
// ===== library types =====

// folder: LIOLink

TYPE "LIOLink_typeDiagnostics"
   STRUCT
      status : Word;   // Status of the Block or error identification when error occurred
      subfunctionStatus : DWord;   // Status or return value of called FB's, FCs and system blocks
      stateNumber : DInt;   // State in the state machine of the block where the error occurred
   END_STRUCT;
END_TYPE

// folder: iJaw

TYPE "UDT_iJawDataRcv"
   STRUCT
      Gauge1 : Word;   // ADC Eingang der Sensorrohdaten (min.: 0 max.: 4096)
      Gauge2 : Word;   // ADC Eingang der Sensorrohdaten (min.: 0 max.: 4096)
      Battery : Byte;   // Rohsignal aktuelle Batteriespannung (min.: 0 .. max.: 157) [V]
      Temperature : Byte;   // Rohsignal Temperatursensor (min.: -40 .. max.: 125) [°C]
      GyroXaxis : Byte;   // Rohsignal Beschleunigungssensor X (min.: -128 .. max.: 127) [g]
      GyroYaxis : Byte;   // Rohsignal Beschleunigungssensor Y (min.: -128 .. max.: 127) [g]
      GyroZaxis : Byte;   // Rohsignal Beschleunigungssensor Z (min.: -128 .. max.: 127) [g]
      Warning : Byte;   // Warnungs-/Fehlercode (Bit0:= Klemmkraft überschritten; Bit1:= Klemmkraft unters
      Force1 : Word;   // Spannkraft Kanal 1 (min.: 0 .. max.: 65,535) [N]
      Force2 : Word;   // Spannkraft Kanal 2 (min.: 0 .. max.: 65,535) [N]
      Reserve1431 : Array[14..31] of Byte;   // Reserve
   END_STRUCT;
END_TYPE

TYPE "UDT_iJawDataSend"
   STRUCT
      nRotSpeedSpindleAct : Int;   // actual rotational speed of the spindle
      pHydCylChamber1Act : Byte;   // actual hydraulic pressure in actuating cylinder chamber for outer clamping
      pHydCylChamber2Act : Byte;   // actual hydraulic pressure in actuating cylinder chamber for outer clamping
      AHydCylChamber1Act : Byte;   // hydraulic area of cylinder chamber for outer clamping
      AHydCylChamber2Act : Byte;   // hydraulic area of cylinder chamber for outer clamping
      Reserve0631 : Array[6..31] of Byte;   // Reserve
   END_STRUCT;
END_TYPE

TYPE "UDT_iJawDataSendUser"
VERSION : 0.1
   STRUCT
      RelCmdSysMode : Bool;   // Trigger sende Kommando change System Mode (see Mode)
      RelCmdTara : Bool;   // Trigger sende Kommando Tara
      RelReadType : Bool;   // Trigger sende Kommando lese iJaw Type
      RelIMA : Bool;   // Trigger sende Kommando IMA
      RelForceTreshold : Bool;   // Trigger sende Kommando Force Treshold
      RelNoiseLevel : Bool;   // Trigger sende Kommando Noise Level
      RelStoreToFlash : Bool;   // Trigger sende Kommando Store to Flash
      NoiseLevel : UInt;   // Höhe der Kraftänderung innerhalb der Samplerate 100Hz, die zur Bestimmung einer Messdatenübertragung neben dem Schwellwert herangezogen wird.
      ForceTreshold : UDInt;   // Schwellwert der Spannkraftsumme die anliegt, um im Mode 2 kontinuierlich Daten zu übertragen
      IMA : USInt;   // Zeitintervall in s, innerhalb der die iJaw spätestens einen neuen Messwert an den Empfänger überträgt
      Mode : Byte;   // Select Mode (0x1 = continuous mode; 0x2 = state dependent mode
      nRotSpeedSpindleAct : Int;   // actual rotational speed of the spindle
      pHydCylChamber1Act : Byte;   // actual hydraulic pressure in actuating cylinder chamber for outer clamping
      pHydCylChamber2Act : Byte;   // actual hydraulic pressure in actuating cylinder chamber for outer clamping
      AHydCylChamber1Act : Byte;   // hydraulic area of cylinder chamber for outer clamping
      AHydCylChamber2Act : Byte;   // hydraulic area of cylinder chamber for outer clamping
   END_STRUCT;
END_TYPE

TYPE "UDT_iJawDataRcvUser"
VERSION : 0.1
   STRUCT
      Gauge1 : UInt;   // ADC Eingang der Sensorrohdaten (min.: 0 max.: 4096)
      Gauge2 : UInt;   // ADC Eingang der Sensorrohdaten (min.: 0 max.: 4096)
      Battery : USInt;   // Rohsignal aktuelle Batteriespannung (min.: 0 .. max.: 157) [V]
      Temperature : SInt;   // Rohsignal Temperatursensor (min.: -40 .. max.: 125) [°C]
      GyroXaxis : SInt;   // Rohsignal Beschleunigungssensor X (min.: -128 .. max.: 127) [g]
      GyroYaxis : SInt;   // Rohsignal Beschleunigungssensor Y (min.: -128 .. max.: 127) [g]
      GyroZaxis : SInt;   // Rohsignal Beschleunigungssensor Z (min.: -128 .. max.: 127) [g]
      Warning : Byte;   // Warnungs-/Fehlercode (Bit0:= Klemmkraft überschritten; Bit1:= Klemmkraft unters
      Force1 : UInt;   // Spannkraft Kanal 1 (min.: 0 .. max.: 65,535) [N]
      Force2 : UInt;   // Spannkraft Kanal 2 (min.: 0 .. max.: 65,535) [N]
      iJawType : String;   // Ausgelesen Typ des iJaws
   END_STRUCT;
END_TYPE

TYPE "UDT_iJawIOFifo"
   STRUCT
      cmd : USInt;   // kommando
      isuCmdData : "UDT_iJawISDUCmdData";
   END_STRUCT;
END_TYPE

TYPE "UDT_iJawISDUCmdData"
TITLE = UDT_iJawISDUCmdData
// Command daten für die isdu / io-link kommunikation
   STRUCT
      execute : Bool;   // Anforderung zum Ausführen der Funktion
      readWrite : Bool;   // FALSE: lesen, TRUE: schreiben
      port : Int;   // Port am IO-Link-Master-Modul
      index : Int;   // Adressparameterindex (IO-Link Device); 0..32767: IOL-D; 65535: Portfunktionen
      subindex : Int;   // Adressparameter Subindex (IO-Link Device); 0: vollständige Aufzeichnung; 1-255: Einzelparameter
      writeLen : Int;   // Länge der Schreibdaten (Nettodaten); 1..232
   END_STRUCT;
END_TYPE

// folder: (top level)

FUNCTION "GetHwDevice" : Int   // FC1, SCL
TITLE = GetHwDevice
{ S7_Optimized_Access := 'TRUE' }
AUTHOR : HeitecAg
VERSION : 0.1
// Ermitteln einer Hardware-Kennung eines DP-Slaves/PROFINET IO-Devices anhand einer E/A-Adresse
   VAR_INPUT
      varEaAdresse : Variant;   // EA-Adresse (E, A, PE, PA) innerhalb eines Moduls.
   END_VAR
   VAR_OUTPUT
      hwDevice : HW_DEVICE;   // Ermittelte Hardware-Kennung eines DP-Slaves/PROFINET IO-Devices
   END_VAR
   VAR_TEMP
      thwAny : HW_ANY;   // Ermittelte Hardware-Kennung (logische Adresse) des EA-Moduls.
      tgeoAdr : GEOADDR;   // Geografische Adresse
   END_VAR
   // Ret_Val : Fehlercode der Anweisungen.
   VAR CONSTANT
      DEF_HE_DEVICE : HW_DEVICE := 0;   // Initalwert für output hw_device
      HWTYPE : UInt := 2;   // Hardwaretyp: 2: IO-Device / DP-Slave
      SLOT : UInt := 0;   // Steckplatz-Nummer
      SUB_SLOT : UInt := 0;   // Nummer des Submoduls. Falls kein Submodul vorhanden ist oder gesteckt werden kann, hat dieser Parameter den Wert "0".
   END_VAR
BEGIN
   REGION BLOCK INFO HEADER
     //==========================================================================================================
     //Title:        GetHwDevice
     //Function:     Ermitteln einer Hardware-Kennung eines DP-Slaves/PROFINET IO-Devices anhand einer E/A-Adresse
     //----------------------------------------------------------------------------------------------------------
     //Change log table:
     //Version       | Date          | Expert in charge      | Changes applied
     //----------------------------------------------------------------------------------------------------------
     //1.0.0         | 26.06.23      | HeitecAg                | First released Version
     //==========================================================================================================
   END_REGION BLOCK INFO HEADER

   #hwDevice := #DEF_HE_DEVICE;

   #GetHwDevice := IO2MOD(ADDR := #varEaAdresse, LADDR => #thwAny);

   IF (#GetHwDevice = 0)THEN
     #GetHwDevice := LOG2GEO(LADDR := #thwAny, GEOADDR := #tgeoAdr);
   END_IF;

   IF (#GetHwDevice = 0) THEN
     #tgeoAdr.HWTYPE := #HWTYPE;
     #tgeoAdr.SLOT := 0;
     #tgeoAdr.SUBSLOT := 0;

     #GetHwDevice := GEO2LOG(GEOADDR := #tgeoAdr, LADDR => #hwDevice);
   END_IF;

   ENO := (#GetHwDevice = 0);
   RETURN;
END_FUNCTION

// folder: LIOLink/S7-1200/1500/Base blocks

FUNCTION_BLOCK "LIOLink_Device"   // FB50004, SCL
TITLE = LIOLink_Device / LIOLINK_DEVICE
{ S7_Optimized_Access := 'TRUE' }
AUTHOR : SIOS
FAMILY : LIOLink
VERSION : 4.0
// Acyclically reads or writes data records from and to IO-Link devices / Funktionsbaustein zum Lesen und Schreiben von azyklischen Daten auf Geräten mit IO-Link, die auf SIMATIC S7-Steuerungen verwendet werden. (früher IO_LINK_CALL)
   VAR_INPUT
      execute : Bool;   // Request to execute function / Anforderung zum Ausführen der Funktion
      hwID : HW_IO;   // Hardware identifier of IO-Link master module or first sub module / Hardware-Kennung des IO-Link-Mastermoduls (Submodul für ET 200eco PN)
      cap : Int;   // Client Access Point (CAP) 0xB400 or 0x00E3 (227) / Client Access Point (CAP); 0xB400 für ET 200eco PN, CM 8x IO-Link, sonst 0xE003 (227)
      readWrite : Bool;   // FALSE: read-mode, TRUE: write-mode / FALSE: lesen, TRUE: schreiben
      port : Int;   // Port on IO-Link master module / Port am IO-Link-Master-Modul
      index : Int;   // Address parameter index (IO-Link device); 0..32767: IOL-D; 65535: port functions / Adressparameterindex (IO-Link Device); 0..32767: IOL-D; 65535: Portfunktionen
      subindex : Int;   // Address parameter subindex (IO-Link device); 0: full record; 1-255: single parameter / Adressparameter Subindex (IO-Link Device); 0: vollständige Aufzeichnung; 1-255: Einzelparameter
      writeLen : Int;   // Length of writing data (net data); 1..232 / Länge der Schreibdaten (Nettodaten); 1..232
      timeout : Time := T#20S;   // Time after which the request is aborted / Zeit, nach der die Anfrage abgebrochen wird
      pollingPeriod : Time := T#100MS;   // Time period of polling
   END_VAR
   VAR_OUTPUT
      done : Bool;   // TRUE: FB processing successfully completed / TRUE: FB-Bearbeitung erfolgreich abgeschlossen
      busy : Bool;   // TRUE: FB is active and new output values can be expected. / TRUE: FB ist aktiv und neue Ausgangswerte sind zu erwarten.
      error : Bool;   // FALSE: No error / TRUE: An error occurred during the execution of the FB. / FALSE: Kein Fehler / TRUE: Bei der Ausführung des FB ist ein Fehler aufgetreten.
      status : Word := 16#7000;   // 16#0000-16#7FFF: Status of the FB / 16#8000-16#FFFF: Error identification (see following table) / 16#0000-16#7FFF: Status des FB / 16#8000-16#FFFF: Fehleridentifikation (siehe folgende Tabelle)
      diagnostics : "LIOLink_typeDiagnostics";   // Diagnostics information of FB / Diagnoseinformationen der FB
      readLen : Int;   // Length of read data record (number of bytes) / Länge des gelesenen Datensatzes (Anzahl Bytes)
   END_VAR
   VAR_IN_OUT
      record : Array[*] of Byte;   // Data area for reading/writing data (max. 232 byte) / Datenbereich zum Lesen/Schreiben von Daten (max. 232 Byte)
   END_VAR
   VAR
      statExecuteOld : Bool;   // Old value of 'execute' input for edge detection / Alter Wert des 'Execute'-Eingangs für Flankenerkennung
      statDone : Bool;   // Static value for output 'done' / Statischer Wert für Ausgang 'done'
      statBusy : Bool;   // Static value for output 'busy' / Statischer Wert für Ausgang 'besetzt'
      statError : Bool;   // Static value for output 'error' / Statischer Wert für Ausgang 'error'
      statStatus : Word := 16#7000;   // Static value for output 'status' / Statischer Wert für Ausgang 'Status'
      statPollingPeriod : Time := T#100MS;   // Static value for input 'pollingPeriod'
      statHwID : HW_IO;   // Static value for input 'hwID' / Statischer Wert für Eingang 'hwID'
      statHwIDprevious : HW_IO;   // Static value for input 'hwID' from the previous execute / Statischer Wert für Eingang 'hwID'
      statReadWrite : Bool;   // Static value for input 'readWrite' / Stativwert für Eingabe 'readWrite'
      statCap : UInt;   // Static value for input 'cap' / Statischer Wert für Eingabe 'cap'
      statTimeout : Time;   // Static value for input 'timeout' / Statischer Wert für Eingang 'timeout'
      statLen : UInt;   // Length of data to be written to device / Länge der Daten, die auf das Gerät geschrieben werden sollen
      statSubfunctionStatus : DWord;   // Status of WRREC/RDREC or error code from IO-Link Master (%W1: IO-Link Master error, %W0: ISDU error) / Status von WRREC/RDREC oder Fehlercode vom IO-Link-Master (%W1: IO-Link-Master-Fehler, %W0: ISDU-Fehler)
      statFBErrorState : DInt;   // State in the state machine of the block where the error occurred / Zustand in der Zustandsmaschine des Blocks, in dem der Fehler aufgetreten ist
      statFBState : DInt := 0;   // State in the state machine of the FB / Zustand in der Zustandsmaschine der FB
      statEmptyDiagnostics : "LIOLink_typeDiagnostics";   // Empty diagnostics information (for initialization purposes only) / Leere Diagnoseinformationen (nur für Initialisierungszwecke)
      instRdRec : RDREC;   // System function "read data record" / Systemfunktion "Datensatz lesen"
      instWrRec : WRREC;   // System function "write data record" / Systemfunktion "Datensatz schreiben"
      instPoll : TP_TIME;   // poll rate read data record / Abfragerate Datensatz lesen
      instMonitor : TON_TIME;   // request monitoring time / Überwachungszeit anfordern
      statRead : Struct   // data area for reading data / Datenbereich zum Lesen von Daten
         header : Struct   // Header
            call : Struct   // header for read/write data record / Header für Datensatz lesen/schreiben
               extFunctionNum : Byte := 16#08;   // extended function number (fix coded 08h) / erweiterte Funktionsnummer (fix codiert 08h)
               port : Byte;   // variable port (user interface) 0...255 / variabler Port (Benutzeroberfläche) 0...255
               fiIndex : Word := 16#FE4A;   // FI index (fix coded 65098) / FI-Index (fix codiert 65098)
            END_STRUCT;
            iolHeader : Struct   // header for IO-Link / Header für IO-Link
               control : Byte;   // RD_WR = 0 = read = Control:=0x03 / / RD_WR = 1 = write = Control:=0x02 / RD_WR = 0 = lesen = Steuerung:=0x03 / / RD_WR = 1 = schreiben = Steuerung:=0x02
               indexHighByte : Byte;   // index of data record 0…32767 (high byte) / Index des Datensatzes 0…32767 (High Byte)
               indexLowByte : Byte;   // index of data record 0…32767 (low byte) / Index des Datensatzes 0…32767 (Low Byte)
               subindex : Byte;   // subindex for data record 0...255 / Subindex für Datensatz 0...255
            END_STRUCT;
         END_STRUCT;
         data : Array[0..231] of Byte;   // Data
      END_STRUCT;
      statWrite : Struct   // data area for writing data / Datenbereich zum Schreiben von Daten
         header : Struct   // Header
            call : Struct   // header for read/write data record / Header für Datensatz lesen/schreiben
               extFunctionNum : Byte := 16#08;   // extended function number (fix coded 08h) / erweiterte Funktionsnummer (fix codiert 08h)
               port : Byte;   // variable port (user interface) 0...255 / variabler Port (Benutzeroberfläche) 0...255
               fiIndex : Word := 16#FE4A;   // FI index (fix coded 65098) / FI-Index (fix codiert 65098)
            END_STRUCT;
            iolHeader : Struct   // header für IO-Link / Header für IO-Link
               control : Byte;   // RD_WR = 0 = read = Control:=0x03 / / RD_WR = 1 = write = Control:=0x02 / RD_WR = 0 = lesen = Steuerung:=0x03 / / RD_WR = 1 = schreiben = Steuerung:=0x02
               indexHighByte : Byte;   // index of data record 0…32767 (high byte) / Index des Datensatzes 0…32767 (High Byte)
               indexLowByte : Byte;   // index of data record 0…32767 (low byte) / Index des Datensatzes 0…32767 (Low Byte)
               subindex : Byte;   // subindex for data record 0...255 / Subindex für Datensatz 0...255
            END_STRUCT;
         END_STRUCT;
         data : Array[0..231] of Byte;   // Data
      END_STRUCT;
   END_VAR
   VAR_TEMP
      tempExecute : Bool;   // Temporary value for input 'execute' / Temporärer Wert für Eingabe 'execute'
      tempHwID : HW_IO;   // Temporary value for input 'hwID'
      tempPort : Int;   // Temporary value for input 'port'
      tempIndex : Int;   // Temporary value for input 'index'
      tempSubindex : Int;   // Temporary value for input 'subindex'
      tempIndexCounter : DInt;   // run tag for counting loops / Run-Tag für Zählschleifen
   END_VAR
   VAR CONSTANT
      MODE_READ : Bool := FALSE;   // Mode to read data / Modus zum Lesen von Daten
      MODE_WRITE : Bool := TRUE;   // Mode to write data / Modus zum Schreiben von Daten
      MAX_PORT : USInt := 63;   // Max. possible port / max. möglichen Hafen
      MAX_INDEX : UInt := 32767;   // Max. possible index / max. möglicher Index
      INDEX_PORT_FUNC : UInt := 65535;   // Index to address port functions / Index zum Adressieren von Portfunktionen
      MAX_SUBINDEX : USInt := 255;   // Max. possible subindex / max. möglicher Subindex
      MAX_DATA : USInt := 232;   // Max. size of data to be transferred / max. Größe der zu übertragenden Daten
      UPPER_LIMIT : DInt := 231;   // Upper limit of data to be transferred / Obergrenze der zu übertragenden Daten
      FB_STATE_NO_PROCESSING : DInt := 0;   // FB state: No processing / FB-Zustand: Keine Verarbeitung
      FB_STATE_WRITE : DInt := 1;   // FB state: Write data record / Datensatz schreiben
      FB_STATE_POLL : DInt := 2;   // FB state: Wait and poll for response / warten und auf Antwort abfragen
      FB_STATE_READ_CAP : DInt := 3;   // FB state: Read cap / CAP lesen
      IOL_HEADER : UInt := 65098;   // Header IO-Link / Kopfzeile IO-Link
      LEN_HEADER : USInt := 8;   // Length of header / Länge des Headers
      CONTROL_WRITE : Byte := 16#02;   // Write data record / Datensatz schreiben
      CONTROL_READ : Byte := 16#03;   // Read data record / Datensatz lesen
      STATUS_EXECUTION_FINISHED : Word := 16#0000;   // Execution finished without errors / Ausführung ohne Fehler beendet
      STATUS_NO_CALL : Word := 16#7000;   // No job being currently processed / Derzeit wird kein Auftrag bearbeitet
      STATUS_FIRST_CALL : Word := 16#7001;   // First call after incoming new job (rising edge 'execute') / Erster Aufruf nach eingehendem neuen Auftrag (steigende Flanke 'execute')
      STATUS_SUBSEQUENT_CALL : Word := 16#7002;   // Subsequent call during active processing without further details / Nachfolgender Aufruf während aktiver Bearbeitung ohne weitere Angaben
      SUB_STATUS_NO_ERROR : Word := 16#0000;   // No error occured in subfunction call / Fehler: falscher Port
      ERR_WRONG_PORT : Word := 16#8201;   // Error: wrong port / Fehler: falscher Index
      ERR_WRONG_INDEX : Word := 16#8202;   // Error: wrong index / Fehler: falscher Subindex
      ERR_WRONG_SUBINDEX : Word := 16#8203;   // Error: wrong subindex / Fehler: falsche Länge für Datensatz schreiben
      ERR_WRONG_LENGTH : Word := 16#8205;   // Error: wrong length for write data record / Fehler: IO-Link-Master hat Fehlercode zurückgegeben, siehe "Diagnose"
      ERR_IO_LINK : Word := 16#8401;   // Error: IO-Link master returned error code, see "diagnostics" / Fehler: Gelesener Datensatz stimmt nicht mit Anfrage überein
      ERR_INCONSISTENT_DATA : Word := 16#8402;   // Error: Read data record doesn't match request / Fehler: Zeitüberschreitung bei Anforderung
      ERR_REQUEST_TIMEOUT : Word := 16#8403;   // Error: Request timed out / Fehler: Aufgrund eines undefinierten Zustands in der Zustandsmaschine
      ERR_UNDEFINED_STATE : Word := 16#8600;   // Error: due to an undefined state in state machine / Fehler: Aufgrund eines undefinierten Zustands in der Zustandsmaschine
      ERR_WRREC : Word := 16#8601;   // Error: WRREC encountered an error, see "diagnostics" / Fehler: WRREC hat einen Fehler festgestellt, siehe "Diagnose"
      ERR_RDREC : Word := 16#8602;   // Error: RDREC encountered an error, see "diagnostics" / Fehler: RDREC hat einen Fehler festgestellt, siehe "Diagnose"
      STATUS_MASK : DWord := 16#00FF_FF00;   // Mask to filter error codes / Maske zum Filtern von Fehlercodes
      STATUS_RESOURCE_BUSY : DWord := 16#0080_C200;   // Status from WRREC/RDREC: Resource is busy / Status von WRREC/RDREC: Ressource ist beschäftigt
      INDEX_CAP_IOLINK : Word := 16#B000;   // Index of the data record for IOLM_Info. Only IO-Link-Masters with CAP=16#B000 support this call. / Index des Datensatzes für IOLM_Info. Nur IO-Link-Master mit CAP=16#B000 unterstützen diesen Aufruf.
      CAP_LEGACY : Word := 16#00E3;   // Siemens (old) Standard CAP: 227 / Siemens (alt) Standard CAP: 227
      CAP_STANDARD : Word := 16#B400;   // IO-Link Standard CAP: 16#B400 / IO-Link-Standard-CAP: 16#B400
      STATUS_RDREC_VALID : Byte := 16#00;   // Status Code of RDREC in cased of no error occurs
      BITMASK_ERR_RDREC_B3 : Byte := 16#DE;   // Status Code of RDREC in case of an error when reading a data record
      BITMASK_ERR_RDREC_B2 : Byte := 16#80;   // Status Code of RDREC in case of an error when reading a data record - Error according to IEC 61158-6
      BITMASK_ERR_RDREC_B1 : Byte := 16#B0;   // Status Code of RDREC in case of an error when reading a data record - invalid index (cap)
   END_VAR
BEGIN
   REGION BLOCK INFO HEADER
       //===============================================================================
       // Siemens / (c)Copyright 2023
       //-------------------------------------------------------------------------------
       // Title:            LIOLink_Device
       // Function:         Acyclically reads or writes data records from and to IO-Link devices
       // Library:          LIOLink
       // Author:           Siemens Industry Online Support
       // Tested with:      CPU 1513-1 PN FW 2.8
       // Engineering:      TIA Portal V16
       // Restrictions:     S7-1200/1500
       // Requirements:     --
       //-------------------------------------------------------------------------------
       // Change log table:
       // Version  | Date       | Expert in charge       | Changes applied
       //----------|------------|------------------------|------------------------------
       // 02.00.00 | 30.09.2013 | Online Support         | First release for TIA Portal V12 SP1 as IO_LINK_CALL
       // 02.01.00 | 14.03.2014 | Online Support         | Upgrade to TIA Portal V13
       //                                                | Upgrade of system function 'WRREC' from V1.0 to V1.1
       // 03.00.00 | 28.02.2015 | SUP Applications       | Upgrade to TIA Portal V13 SP1
       //                                                | Renamed FB to IO_LINK_DEVICE 
       // 03.01.00 | 15.09.2015 | SUP Applications       | Change of #IOL_INDEX AND #Port lower boundry to 0 and improved behaviour when called in cyclic OBs with > 100 ms
       // 04.00.00 | 01.09.2020 | Online Support         | Implemented Programming styleguide for S7-1200/1500 and PLCopen
       //                                                | Renamed FB to LIOLink_Device 
       // 05.00.00 | 28.02.2023 | SUP SPH                | Added Polling Time as predefined input
       //                                                | #record is changed to a variable array (Array[*])
       //                                                | Changed CAP as predefined variable, added functionality to automatically find CAP of IO-Link-Masters from SIEMENS                                               
       //===============================================================================
   END_REGION

   REGION TRIGGERING
       #tempExecute := #execute; // Work with temporary value / create process image

       IF (#tempExecute = TRUE) AND (#statExecuteOld = FALSE) // Check if FB is triggered
           AND (#statStatus = #STATUS_NO_CALL)
       THEN
           REGION Initialize data
               // First call; initialize FB
               #statDone := FALSE;
               #statBusy := TRUE;
               #statError := FALSE;
               #statStatus := #STATUS_FIRST_CALL;
               #statSubfunctionStatus := #SUB_STATUS_NO_ERROR;
               #statFBErrorState := 0;
               #diagnostics := #statEmptyDiagnostics;
               #readLen := 0;

               // Initialize data area
               #statRead.header."call"."port" := 16#0;
               #statRead.header.iolHeader.indexLowByte := 16#0;
               #statRead.header.iolHeader.indexHighByte := 16#0;
               #statRead.header.iolHeader.subindex := 16#0;
               #tempIndexCounter := 0; // initialize loop counter      
               FOR #tempIndexCounter := 0 TO #UPPER_LIMIT DO
                   #statWrite.data[#tempIndexCounter] := 16#0;
                   #statRead.data[#tempIndexCounter] := 16#0;
               END_FOR;
           END_REGION

           REGION Save inputs
               // Copy input variables to temporary variables
               #tempHwID := #hwID;
               #statReadWrite := #readWrite;
               #statTimeout := #timeout;
               #statPollingPeriod := #pollingPeriod;
               #tempPort := #port;
               #tempIndex := #index;
               #tempSubindex := #subindex;
           END_REGION

           REGION Build header
               // setup call header
               #statWrite.header."call"."port" := INT_TO_BYTE(#tempPort);

               // setup IOL header 
               #statWrite.header.iolHeader.indexLowByte := INT_TO_BYTE(#tempIndex);
               #statWrite.header.iolHeader.indexHighByte := INT_TO_BYTE(SHR(IN := #tempIndex, N := 8));
               #statWrite.header.iolHeader.subindex := INT_TO_BYTE(#tempSubindex);

               // BODY (data max. 232 Byte, Array 0..231 of Byte) 
               IF #statReadWrite = #MODE_WRITE THEN // Write data record requested, copy data from "record"
                   #statWrite.header.iolHeader.control := #CONTROL_WRITE;
                   #statLen := INT_TO_UINT(#writeLen) + #LEN_HEADER; // data length header + data = IO-Link write data record
                   // copy "record" to working area
                   FOR #tempIndexCounter := 0 TO #writeLen - 1 DO
                       #statWrite.data[#tempIndexCounter] := #record[#tempIndexCounter];
                   END_FOR;
               ELSE // Read data record requested
                   // Empty record array
                   FILL_BLK(IN := 16#0,
                            COUNT := #MAX_DATA,
                            OUT => #record[0]);

                   #statWrite.header.iolHeader.control := #CONTROL_READ;
                   #statLen := #LEN_HEADER; // data length only header = IO-Link read data record
               END_IF;
           END_REGION

           REGION Check parameters
               // Check parameters
               IF (#tempPort < 0) OR (#tempPort > #MAX_PORT) THEN
                   #statStatus := #ERR_WRONG_PORT;
               ELSIF (#tempIndex < 0) OR (#tempIndex > #MAX_INDEX AND #tempIndex <> #INDEX_PORT_FUNC) THEN
                   #statStatus := #ERR_WRONG_INDEX;
               ELSIF (#tempSubindex < 0) OR (#tempSubindex > #MAX_SUBINDEX) THEN
                   #statStatus := #ERR_WRONG_SUBINDEX;
               ELSIF #statReadWrite = #MODE_WRITE AND (#writeLen < 1 OR #writeLen > #MAX_DATA) THEN
                   #statStatus := #ERR_WRONG_LENGTH;
               END_IF;
               //save the hwID from the previous execute
               #statHwIDprevious := #statHwID;

               IF #statStatus = #STATUS_FIRST_CALL THEN // Parameters OK
                   IF #cap <> 0 THEN
                       #statCap := INT_TO_UINT(#cap);
                       #statFBState := #FB_STATE_WRITE;
                   ELSIF (#statCap <> WORD_TO_UINT(#CAP_STANDARD) AND #statCap <> WORD_TO_UINT(#CAP_LEGACY)) OR (#statHwIDprevious <> #tempHwID) THEN // check if new device is connected => hwID changed
                       #statFBState := #FB_STATE_READ_CAP;
                   ELSE
                       #statFBState := #FB_STATE_WRITE;
                   END_IF;
               END_IF;
               // save current hwID
               #statHwID := #tempHwID;
           END_REGION

       ELSIF (#statStatus = #STATUS_FIRST_CALL) THEN
           #statStatus := #STATUS_SUBSEQUENT_CALL;
       END_IF;

       // Edge detection 'execute' input
       #statExecuteOld := #tempExecute;
   END_REGION TRIGGERING

   REGION STATE_MACHINE
       CASE #statFBState OF
           #FB_STATE_NO_PROCESSING:
               REGION no processing
                   ; // No processing active
               END_REGION no processing    

           #FB_STATE_READ_CAP:
               REGION get cap
                   // To find out CAP of IO-Link Master, data record with Index 16#B000 is read. If this reading was successful
                   // then CAP is 16#B400 (based on IO-Link Standard). If the reading was not successful and the status of RDREC
                   // is 16#DE80_B0xx, then CAP is 16#00E3 (227, based on Siemens Old Standard for IO-Link Masters).

                   #instRdRec(RECORD := #statRead);

                   IF (#instRdRec.BUSY = FALSE) THEN
                       IF (#instRdRec.VALID = FALSE) AND (#instRdRec.ERROR = FALSE) THEN
                           IF #instRdRec.REQ = FALSE THEN
                               // call read record with Index 16#B000
                               #instRdRec.REQ := true;
                               #instRdRec.ID := #statHwID;
                               #instRdRec.INDEX := WORD_TO_UINT(#INDEX_CAP_IOLINK);
                               #instRdRec.MLEN := 0;
                               #statFBState := #FB_STATE_READ_CAP;
                           END_IF;
                       ELSIF #instRdRec.VALID = TRUE THEN
                           #instRdRec.REQ := FALSE;
                           // if status of RDREC is valid then CAP is 16#B400 (CAP_STANDARD)
                           IF #instRdRec.STATUS.%B3 = #STATUS_RDREC_VALID THEN
                               #statCap := WORD_TO_UINT(#CAP_STANDARD);
                           END_IF;
                           #statFBState := #FB_STATE_WRITE;
                       ELSE
                           // if RDREC is in error state and Status is 16#DE80_B0xx then CAP is 227 (CAP_Legacy)
                           IF (#instRdRec.STATUS.%B3 = #BITMASK_ERR_RDREC_B3) AND (#instRdRec.STATUS.%B2 = #BITMASK_ERR_RDREC_B2) AND (#instRdRec.STATUS.%B1 = #BITMASK_ERR_RDREC_B1) THEN
                               #statCap := WORD_TO_UINT(#CAP_LEGACY);
                               #statFBState := #FB_STATE_WRITE;
                           ELSE
                               #statStatus := #ERR_RDREC;
                               #statSubfunctionStatus := #instRdRec.STATUS;
                               #statCap := 0; //clear CAP if an error occurs
                           END_IF;
                       END_IF;
                   ELSE
                       #instRdRec.REQ := FALSE;
                       IF #instRdRec.ERROR = TRUE THEN
                           #statStatus := #ERR_RDREC;
                           #statSubfunctionStatus := #instRdRec.STATUS;
                           #statCap := 0; //clear CAP if an error occurs
                       END_IF;
                   END_IF;

                   #instRdRec(RECORD := #statRead);
               END_REGION

           #FB_STATE_WRITE:
               REGION write
                   // To read data records, the IO-Link master modules needs to know which port is required. Therefore it is necessary
                   // to send at first a request via write data record (header, 8 byte). As response the IO-Link master module will 
                   // send the required data record.

                   #instWrRec(REQ := TRUE,
                              ID := #statHwID,
                              INDEX := #statCap,
                              LEN := #statLen,
                              RECORD := #statWrite);

                   IF #instWrRec.ERROR THEN
                       IF (#instWrRec.STATUS AND #STATUS_MASK) = #STATUS_RESOURCE_BUSY THEN
                           #instWrRec(REQ := FALSE); // Reset requeset
                       ELSE
                           #statStatus := #ERR_WRREC;
                           #statSubfunctionStatus := #instWrRec.STATUS;
                           #statFBErrorState := #statFBState;
                       END_IF;
                   ELSIF #instWrRec.DONE = TRUE THEN
                       #instWrRec(REQ := FALSE); // Reset requeset

                       #statFBState := #FB_STATE_POLL;
                   END_IF;
               END_REGION write

           #FB_STATE_POLL: // wait and poll for response
               REGION poll
                   #instPoll(IN := TRUE,
                             PT := #statPollingPeriod);

                   // read data record on falling edge
                   #instRdRec(REQ := NOT #instPoll.Q,
                              ID := #statHwID,
                              INDEX := #statCap,
                              MLEN := 0, // read all data available,
                              RECORD := #statRead);

                   IF #instRdRec.ERROR = TRUE THEN
                       IF (#instRdRec.STATUS AND #STATUS_MASK) = #STATUS_RESOURCE_BUSY THEN
                           // Reset requests and try again
                           #instPoll(IN := FALSE,
                                     PT := #statPollingPeriod);

                           #instRdRec(REQ := FALSE,
                                      RECORD := #statRead);
                       ELSE
                           #statStatus := #ERR_RDREC;
                           #statSubfunctionStatus := #instRdRec.STATUS;
                           #statFBErrorState := #statFBState;
                       END_IF;
                   ELSIF #instRdRec.VALID THEN
                       IF // check the response wether it matches the request (compare PORT, INDEX and SUBINDEX)
                           (#statWrite.header."call"."port" <> #statRead.header."call"."port")
                           OR (#statWrite.header.iolHeader.indexHighByte <> #statRead.header.iolHeader.indexHighByte)
                           OR (#statWrite.header.iolHeader.indexLowByte <> #statRead.header.iolHeader.indexLowByte)
                           OR (#statWrite.header.iolHeader.subindex <> #statRead.header.iolHeader.subindex)
                       THEN // read data record doesn't match the request
                           #statStatus := #ERR_INCONSISTENT_DATA;  // output status no consistent data
                       ELSIF #statRead.header.iolHeader.control = B#16#80 THEN // check the response for IO-Link errors
                           // State 0x80 = IOL_CALL_RES PDU shows IO-Link error detect
                           #statStatus := #ERR_IO_LINK;
                           #statSubfunctionStatus.%B3 := #statRead.data[0]; // IO-Link master error code
                           #statSubfunctionStatus.%B2 := #statRead.data[1]; // IO-Link master error code
                           #statSubfunctionStatus.%B1 := #statRead.data[2]; // ISDU error code
                           #statSubfunctionStatus.%B0 := #statRead.data[3]; // ISDU additional code
                           #statFBErrorState := #statFBState;
                       ELSE // read data is valid
                           IF #statReadWrite = #MODE_READ THEN
                               #readLen := UINT_TO_INT(#instRdRec.LEN - #LEN_HEADER);
                               // only data will be output
                               FOR #tempIndexCounter := 0 TO UINT_TO_INT(#instRdRec.LEN - #LEN_HEADER - 1) DO
                                   #record[#tempIndexCounter] := #statRead.data[#tempIndexCounter];
                               END_FOR;
                           END_IF;

                           // Reset requests
                           #instRdRec(REQ := FALSE,
                                      RECORD := #statRead);

                           #instPoll(IN := FALSE,
                                     PT := #statPollingPeriod);

                           #statStatus := #STATUS_EXECUTION_FINISHED;  // request finished
                       END_IF;
                   END_IF;
               END_REGION poll

           ELSE // Undefined state in state machine reached
               REGION undefined state
                   #statStatus := #ERR_UNDEFINED_STATE;
               END_REGION undefined state no relevant case, ready for new request
       END_CASE;
   END_REGION

   REGION MONITORING
       #instMonitor(IN := #statBusy,
                    PT := #statTimeout);

       IF #instMonitor.Q THEN
           #statStatus := #ERR_REQUEST_TIMEOUT; // request time out
       END_IF;
   END_REGION

   REGION OUTPUTS
       // Write outputs
       IF (#statStatus = #STATUS_EXECUTION_FINISHED) AND (#statDone = FALSE) THEN // Execution finished without errors, available only for one cycle
           REGION execution finished
               #statDone := TRUE;
               #statBusy := FALSE;
               #statError := FALSE;
               // execution aborted --> set state no processing
               #statFBState := #FB_STATE_NO_PROCESSING;
           END_REGION execution finished

       ELSIF (#statStatus.%X15 = TRUE) AND (#statError = FALSE) THEN // Error occurred (#statStatus is 16#8000 to 16#FFFF), Error status is true only for one cycle (the second last cycle)
           REGION error occured
               #statDone := FALSE;
               #statBusy := FALSE;
               #statError := TRUE;
               #statCap := 0; //Reset statcap, if error occurs, get cap has to be performed again
               // Write diagnostics
               #diagnostics.status := #statStatus;
               #diagnostics.subfunctionStatus := #statSubfunctionStatus;
               #diagnostics.stateNumber := #statFBErrorState;
               // Call instructions with FALSE to be ready for next job
               #instWrRec(REQ := FALSE);

               #instRdRec(REQ := FALSE,
                          RECORD := #statRead);

               #instPoll(IN := FALSE,
                         PT := #statPollingPeriod);

               // execution aborted --> set state no processing
               #statFBState := #FB_STATE_NO_PROCESSING;
           END_REGION error occured

       ELSIF (#tempExecute = FALSE) AND ((#statDone = TRUE) OR (#statError = TRUE)) THEN // Reset outputs, Last cycle
           REGION execute reset
               #statDone := FALSE;
               #statBusy := FALSE;
               #statError := FALSE;
               #statStatus := #STATUS_NO_CALL;
               #readLen := 0;
           END_REGION execute reset
       END_IF;

       REGION write static values to outputs
           #done := #statDone;
           #busy := #statBusy;
           #error := #statError;
           #status := #statStatus;
           //ENO := NOT #statError;
       END_REGION write static values to outputs
   END_REGION OUTPUTS
END_FUNCTION_BLOCK

// folder: iJawBib

FUNCTION_BLOCK "SendRcv_iJaw_2TH"   // FB3, SCL
TITLE = SendRcv_iJaw
{ S7_Optimized_Access := 'TRUE' }
AUTHOR : HeitecAg
VERSION : 0.1
// Kommunikation mit den iJaw Backen mittels IO-LInk und Profinet
   VAR_INPUT
      iLADDR_TigoMaster : HW_DEVICE;   // HW-Device aus Hardwarekonfiguration TigoMaster
      iPN_Act : Bool;   // De-/Aktivierung Profinetteilnehmer 1= Aktivieren 0= Deaktivieren
      iCpuRestart : Bool;   // Restartmerker der SPS Wenn keiner vorhanden dann mit False besetzten.
      iAck_Fehler_IoLinkKom : Bool;   // Quitterung des Kommunikationsfehlers.(Sende-/ Lese Aufträge werden danach erneut gestartet)
      iResetIoLinkKom : Bool;   // Reset der LIO-Link kommunikation (Alle Sende-/ Lese Aufträge werden gelöscht)
      iTime_PnIoRyd : Time;   // Zeit zum Hochlauf des Bussystems / des TigoMasters (Vermeidung von Lesefehlern)
      iIJawAktiv_iJaw1 : Bool;   // iJaw 1 ist aktiv & vorhanden
      iIJawAktiv_iJaw2 : Bool;   // iJaw 2 ist aktiv & vorhanden
      iIJawAktiv_iJaw3 : Bool;   // iJaw 3 ist aktiv & vorhanden
      iIJawAktiv_iJaw4 : Bool;   // iJaw 4 ist aktiv & vorhanden
      iIJawAktiv_iJaw5 : Bool;   // iJaw 5 ist aktiv & vorhanden
      iIJawAktiv_iJaw6 : Bool;   // iJaw 6 ist aktiv & vorhanden
      iIJawAktiv_iJaw7 : Bool;   // iJaw 7 ist aktiv & vorhanden
      iIJawAktiv_iJaw8 : Bool;   // iJaw 7 ist aktiv & vorhanden
      iFreeIsduCmd : "UDT_iJawISDUCmdData";   // Freier ISDU-Auftrag
      iFreeIsduSendData : Array[0..#LAENGE_IOLINK_RECORD] of Byte;   // Datenbereich zum Schreiben für den freien ISDU-Auftrag
      iUserDaten_iJaw1 : "UDT_iJawDataSendUser";   // Sendedaten PLC --> iJaw 01
      iUserDaten_iJaw2 : "UDT_iJawDataSendUser";   // Sendedaten PLC --> iJaw 02
      iUserDaten_iJaw3 : "UDT_iJawDataSendUser";   // Sendedaten PLC --> iJaw 03
      iUserDaten_iJaw4 : "UDT_iJawDataSendUser";   // Sendedaten PLC --> iJaw 04
      iUserDaten_iJaw5 : "UDT_iJawDataSendUser";   // Sendedaten PLC --> iJaw 05
      iUserDaten_iJaw6 : "UDT_iJawDataSendUser";   // Sendedaten PLC --> iJaw 06
      iUserDaten_iJaw7 : "UDT_iJawDataSendUser";   // Sendedaten PLC --> iJaw 07
      iUserDaten_iJaw8 : "UDT_iJawDataSendUser";   // Sendedaten PLC --> iJaw 08
   END_VAR
   VAR_OUTPUT
      oError : Bool;   // Fehler bei der Abarbeitung des Bausteines
      oPnTeilAkt : Bool;   // Status des Profinetteilnehmer 1= Teilnehmer aktiv 0= Teilnehmer deaktiviert
      oIoLinkRdy : Bool;   // Ío link kommunikation bereit zum senden / empfangen
      oIoLinkBusy : Bool;   // Ío link kommunikation beschäftig
      oIoLinkError : Bool;   // Ío link kommunikation fehlerhaft
      oFreeIsduCmdFertig : Bool;   // Freier ISDU-Auftrag erfolgreich abgeschlossen
      oFreeIsduCmdDataBereit : Bool;   // Empfange ISDU-Daten liegen bereit
      oFreeIsduRcvData : Array[0..#LAENGE_IOLINK_RECORD] of Byte;   // Empfange ISDU-Daten
      oUserDaten_iJaw1 : "UDT_iJawDataRcvUser";   // Empfangsdaten PLC <-- iJaw 01
      oUserDaten_iJaw2 : "UDT_iJawDataRcvUser";   // Empfangsdaten PLC <-- iJaw 02
      oUserDaten_iJaw3 : "UDT_iJawDataRcvUser";   // Empfangsdaten PLC <-- iJaw 03
      oUserDaten_iJaw4 : "UDT_iJawDataRcvUser";   // Empfangsdaten PLC <-- iJaw 04
      oUserDaten_iJaw5 : "UDT_iJawDataRcvUser";   // Empfangsdaten PLC <-- iJaw 05
      oUserDaten_iJaw6 : "UDT_iJawDataRcvUser";   // Empfangsdaten PLC <-- iJaw 06
      oUserDaten_iJaw7 : "UDT_iJawDataRcvUser";   // Empfangsdaten PLC <-- iJaw 07
      oUserDaten_iJaw8 : "UDT_iJawDataRcvUser";   // Empfangsdaten PLC <-- iJaw 08
   END_VAR
   VAR
      xlocalInit : Bool := TRUE;   // lokale initalisierung
      xlocalError : Bool;   // lokale Fehler ist aufgetreten
      xMin1iJawVorh : Bool;   // mindesten eine iJaw konfiguriert
      xSchrittketteTimeOut : Bool;   // schrittkette hat ein timeout fehler
      xSchrittErsterZyklus : Bool;   // flanke erster zyklus im schritt
      xFehlerSchrittZeitUeberwachung : Bool;   // fehler schrittzeitüberwachung
      xlocalIoLinkRdy : Bool;   // Ío link kommunikation bereit zum senden / empfangen
      xlocalIoLinkBusy : Bool;   // Ío link kommunikation beschäftig
      xlocalIoLinkError : Bool;   // Ío link kommunikation fehlerhaft
      xlocalFreeIsduCmdFertig : Bool;   // Freier ISDU-Auftrag erfolgreich abgeschlossen
      xlocalFreeIsduCmdDataBereit : Bool;   // Empfange ISDU-Daten liegen bereit
      dtCpuSystemDatumZeit : Date_And_Time;   // datum und uhrzeit cpu
      todCpuSystemZeit : Time_Of_Day;   // zeit des tages cpu
      tSchrittZeitVortag : Time;   // schrittzeit vom vortag
      tCpuSystemZeit : Time;   // zeit der cpu
      tStartZeitSchritt : Time;   // startzeit des aktuellen schrittes
      tAktuelleSchrittzeit : Time;   // aktuelle schrittzeit
      tMinSchrittZeit : Time;   // minimum zeit des aktiven schrittes
      tMaxSchrittZeit : Time;   // maximum zeit des aktiven schrittes (T#0ms = schrittzeit überwachung deaktiviert)
      fpCpuRestart : R_TRIG;   // flanke positiv cpu wurde neugestartet
      fpResetIoLink : R_TRIG;   // flanke positiv trigger reset io-link kommunikation / löschen desfifo puffers
      fpPnIOAktiv : R_TRIG;   // flanke positiv profinetteilnehmer ist aktiviert
      fpPnIOInAktiv : R_TRIG;   // flanke positiv profinetteilnehmer ist deaktiviert
      arrIJawVorhandenAktiv : Array[1..#MAX_ANZAHL_IJAWS] of Bool;   // speicher der überprüfung von vorhandenen und aktiven iJaws
      iRetRcvData : Int;   // retval Profinetdaten lesen
      iRetSer : Int;   // retval Profinetdaten umladen
      iRetSendData : Int;   // retval Profinetdaten schreiben
      iRetValCpuZeitLesen : Int;   // rückgabewert lesen der cpu zeit
      iRetValLog2Geo : Int;   // rückgabewert LOG2GEO
      iRetValWriteBig : Int;   // rückgabewert WRITE_BIG
      iRetValGeoLog : Array[1..#MAX_HW_SLOTS] of Int;   // rückgabewert GEO_LOG
      diAkuelleSchrittnr : DInt := 0;   // aktuelle Schrittnummer
      diAlteSchrittnr : DInt;   // alte Schrittnummer
      diUrAlteSchrittnr : DInt;   // uralte Schrittnummer
      usiLetzterFiFoEintrag : USInt;   // speicher des letzten eintrags im FIFO-Puffer
      tonPNHochlaufzeit : TON_TIME;   // verzögerung profinet hochlaufzeit
      strcDeaktAkt : Struct   // speicher an/abmelden profinet teilnehmer
         ReqAkt : Bool;
         ReqDeak : Bool;
         IstAkt : Bool;
         IstDeak : Bool;
         ModNr : USInt;
         busy : Bool;
         Ret_Val : Int;
         ChangeRequest_old : Bool;
         FP_Changerequest : Bool;
      END_STRUCT;
      strcIoLinkSignale : Struct   // io-link device variablen
         in : Struct
            execute : Bool;   // Anforderung zum Ausführen der Funktion
            hwID : HW_IO;   // Hardware-Kennung des IO-Link-Mastermoduls (Submodul für ET 200eco PN)
            cap : Int;   // Client Access Point (CAP); 0xB400 für ET 200eco PN, CM 8x IO-Link, sonst 0xE003 (227)
            readWrite : Bool;   // FALSE: lesen, TRUE: schreiben
            port : Int;   // Port am IO-Link-Master-Modul
            index : Int;   // Adressparameterindex (IO-Link Device); 0..32767: IOL-D; 65535: Portfunktionen
            subindex : Int;   // Adressparameter Subindex (IO-Link Device); 0: vollständige Aufzeichnung; 1-255: Einzelparameter
            writeLen : Int;   // Länge der Schreibdaten (Nettodaten); 1..232
            timeout : Time := T#20S;   // Zeit, nach der die Anfrage abgebrochen wird
            pollingPeriod : Time := T#100MS;
         END_STRUCT;
         out : Struct
            done : Bool;   // TRUE: FB-Bearbeitung erfolgreich abgeschlossen
            busy : Bool;   // TRUE: FB ist aktiv und neue Ausgangswerte sind zu erwarten.
            error : Bool;   // FALSE: Kein Fehler / TRUE: Bei der Ausführung des FB ist ein Fehler aufgetreten.
            status : Word;   // 16#0000-16#7FFF: Status des FB / 16#8000-16#FFFF: Fehleridentifikation (siehe folgende Tabelle)
            diagnostics : "LIOLink_typeDiagnostics";   // Diagnoseinformationen der FB
            readLen : Int;   // Länge des gelesenen Datensatzes (Anzahl Bytes)
         END_STRUCT;
         record : Array[0..#LAENGE_IOLINK_RECORD] of Byte;   // Datenbereich zum Lesen/Schreiben von Daten (max. 232 Byte)
      END_STRUCT;
      wErrorW0 : Word;   // fehler status io-link device word 0
      wErrorW1 : Word;   // fehler status io-link device word 1
      instLIOLinkDev : "LIOLink_Device";
      fpTriggerFreeISDU : R_TRIG;   // flanken positiv trigger io-link freier isdu auftrag
      fpTriggerTara : Array[1..#MAX_ANZAHL_IJAWS] of R_TRIG;   // flanken positiv trigger io-link kommando tara
      fpTriggerSySMode : Array[1..#MAX_ANZAHL_IJAWS] of R_TRIG;   // flanken positiv trigger io-link kommando sys-mode
      fpTriggerReadType : Array[1..#MAX_ANZAHL_IJAWS] of R_TRIG;   // flanken positiv trigger io-link kommando sys-mode
      fpTriggerIMA : Array[1..#MAX_ANZAHL_IJAWS] of R_TRIG;   // flanken positiv trigger io-link kommando sys-mode
      fpTriggerForceThreshold : Array[1..#MAX_ANZAHL_IJAWS] of R_TRIG;   // flanken positiv trigger io-link kommando sys-mode
      fpTriggerNoiseLevel : Array[1..#MAX_ANZAHL_IJAWS] of R_TRIG;   // flanken positiv trigger io-link kommando sys-mode
      fpTriggerStoreToFlash : Array[1..#MAX_ANZAHL_IJAWS] of R_TRIG;   // flanken positiv trigger io-link kommando sys-mode
      fifoPuffer : Array[1..#MAX_FIFO_IDX] of "UDT_iJawIOFifo";   // fifo-puffer
      hwAnySubSlotsTigoMaster2Th : Array[1..#MAX_HW_SLOTS] of HW_ANY;   // hardware subslot informationen tigomaster 2th
      strIJawType : Array[1..#MAX_ANZAHL_IJAWS] of String;   // Typ des gewähle iJaws
      recordDataFreeISDU : Array[0..#LAENGE_IOLINK_RECORD] of Byte;   // Datenbereich zum Lesen/Schreiben von Daten (max. 232 Byte)
   END_VAR
   VAR_TEMP
      txFPCpuHochlauf : Bool;   // flanke cpu hochlauf / init
      txAktNächstenSchritt : Bool;   // aktiviere nächsten schritt
      tdiI : DInt;   // iterator
      tdiO : DInt;   // iterator
      tempPosSer : DInt;   // pos für de-/serialize
      tempSchrittNr : DInt;   // nächste schrittnummer
      tempHwAny : HW_ANY;   // temporärer hw any
      tempInitRecord : Array[0..#LAENGE_IOLINK_RECORD] of Byte;   // ablesen die Recordaten
      tempHwInfoTigoMaster2Th : GEOADDR;   // hardware slot informationen tigomaster 2th
      tempResetFifo : "UDT_iJawIOFifo";   // reset fifo eintrag
      tempRcvUserdaten : Array[1..#MAX_ANZAHL_IJAWS] of "UDT_iJawDataRcvUser";   // temporär empfangene user-daten
      tempSendUserDaten : Array[1..#MAX_ANZAHL_IJAWS] of "UDT_iJawDataSendUser";   // temporäre user-sende daten
      tempSendDaten : "UDT_iJawDataSend";   // temporär empfangene daten aller iJaw's
      tempRcvEinzelDaten : "UDT_iJawDataRcv";   // temporär empfangene daten einer iJaw
      tempRcvRohDaten : Array[1..#LAENGE_RCV_DATEN] of Byte;   // temporär empfangene roh daten einer iJaw
      tempIJawAktiv : Array[1..#MAX_ANZAHL_IJAWS] of Bool;   // speicher der überprüfung von aktiven iJaws
   END_VAR
   VAR CONSTANT
      MAX_ANZAHL_IJAWS : USInt := 8;   // maximale anzahl von ijaws
      LAENGE_RCV_DATEN : DInt := 33;   // länge von empfangsdaten
      LAENGE_SEND_DATEN : DInt;   // länge von sende daten
      LAENGE_IOLINK_RECORD : DInt := 231;   // länge von io-link record daten
      CAP_IOLINK : Int := 16#B400;   // Client Access Point (CAP); 0xB400 für ET 200eco PN, CM 8x IO-Link, sonst 0xE003 (227)
      CMD_IDLE : USInt := 0;   // kein kommando steht an
      CMD_TARA : USInt := 1;   // Kommando send tara
      CMD_CHANGE_SYSMODE : USInt := 2;   // Kommando send change system mode
      CMD_READ_TYPE : USInt := 3;   // Kommando send read iJaw type
      CMD_APPLICATION_IMA : USInt := 4;   // Kommando send app ima
      CMD_FORCE_TRESHOLD : USInt := 5;   // Kommando send force treshshold
      CMD_NOISE_LEVEL : USInt := 6;   // Kommando send noise level
      CMD_STORE_TO_FLASH : USInt := 7;   // Kommando send strore to flash
      CMD_FREE_ISDU : USInt := 8;   // Kommando freier isdu auftrag
      IDX_CMD_TARA : Int := 518;   // io-link idx cmd tara
      IDX_CMD_SYSMODE : Int := 518;   // io-link idx cmd system mode
      IDX_CMD_READ_TYPE : Int := 518;   // io-link idx cmd system mode
      IDX_CMD_APPLICATION_IMA : Int := 518;   // io-link idx cmd application IMA
      IDX_CMD_FORCE_THRESHOLD : Int := 516;   // io_link idx cmd force treshold
      IDX_CMD_NOISE_LEVEL : Int := 518;   // io_link idx cmd noise level
      IDX_CMD_STORE_TO_FLASH : Int := 517;   // io_link idx cmd store to flash
      SUB_IDX_CMD_TARA : Int := 15;   // io-link sub idx cmd tara
      SUB_IDX_CMD_SYSMODE : USInt := 4;   // io-link sub idx cmd system mode
      SUB_IDX_CMD_READ_TYPE : USInt := 9;   // io-link sub idx cmd read type
      SUB_IDX_CMD_APPLICATION_IMA : Int := 12;   // io-link sub idx cmd application IMA
      SUB_IDX_CMD_FORCE_TRESHOLD : Int := 1;   // io-link sub idx cmd force treshold
      SUB_IDX_CMD_NOISE_LEVEL : Int := 11;   // io-link sub idx cmd noise level
      SUB_IDX_SCMD_TORE_TO_FLASH : Int := 1;   // io-link sub idx store to flash
      RECORD_DATA_TARA : Byte := 1;   // io-link reocrd daten tara
      RECORD_STORE_TO_FLASH : Byte := 1;   // io-link reocrd daten store to flash
      READ : Bool := FALSE;   // io-link Daten lesen
      WRITE : Bool := TRUE;   // io-link Daten schreiben
      SCHRITT_RESET : DInt := 0;   // schrittnummer check io-link kommuikations
      SCHRITT_CHECK_RDY : DInt := 1;   // schrittnummer check io-link kommuikations
      SCHRITT_HOME : DInt := 2;   // schrittnummer home / warte auf befehel
      SCHRITT_SEND_CMD : DInt := 3;   // schrittnummer sende tara
      SCHRITT_WARTE_AUF_DONE : DInt := 11;   // schrittnummer warte auf auftrag abgeschlossen
      SCHRITT_BEARBEITE_FIFO : DInt := 12;   // schrittnummer bearbeite fifo-puffer
      SCHRITT_FEHLER : DInt := 13;   // schrittnummer fehler
      MAX_FIFO_IDX : USInt := 255;   // maximale fifo einträge
      DEF_TIME_OF_DAY : Time_Of_Day := TOD#00:00:00;   // tages start zeit
      MAX_TIME : Time := T#+24d_20h_31m;   // maximal zeit im timeformat
      IDX_FIFO_LESE_INDEX : USInt := 1;   // index des fifo eintrags zum lesen des auftrags
      DEAK_SCHRITT_ZEIT_UEBERW : Time := T#0ms;   // deaktivierung der schrittzeit überwachung
      MAX_HW_SLOTS : DInt := 9;   // maximal slots in hw (8 ijwas + io-link master)
      KEIN_FEHLER : Int := 0;   // kein fehler aufgetreten
      DEF_HW_ANY : HW_ANY := 0;   // default hw any wert
      SLOT_IDX_MAIN_MODUL_2TH : Int := 1;   // hw slot index des 16 port io-link wirles masters
      HW_IDX_IO_LINK_MASTER : Int := 1;   // array index vom io link master
      HW_IDX_IJAW_1 : Int := 2;   // array index von ijaw 1
      HW_IDX_IJAW_2 : Int := 3;   // array index von ijaw 2
      HW_IDX_IJAW_3 : Int := 4;   // array index von ijaw 3
      HW_IDX_IJAW_4 : Int := 5;   // array index von ijaw 4
      HW_IDX_IJAW_5 : Int := 6;   // array index von ijaw 5
      HW_IDX_IJAW_6 : Int := 7;   // array index von ijaw 6
      HW_IDX_IJAW_7 : Int := 8;   // array index von ijaw 7
      HW_IDX_IJAW_8 : Int := 9;   // array index von ijaw 8
      LEER_STRING : String;   // leere string zum ablöchen
      CNT_CONV_STRING : UInt := 128;   // Anzahl der zu kopierenden Zeichen. Bei "0" werden alle Zeichen kopiert.
      P_CHAR_CONV_STRING : DInt := 0;   // Position im Array of (W)CHAR / BYTE / WORD, ab der die Zeichen kopiert werden.
   END_VAR
   // // iFreeIsduCmd.port : Port am IO-Link-Master-Modul (Nummer der iJaw 1-8)
BEGIN
   REGION BLOCK INFO HEADER
     //==========================================================================================================
     //Title:        SendRcv_iJaw
     //Function:     Kommunikation mit den iJaw Backen mittels IO-LInk und Profinet (2TH)
     //----------------------------------------------------------------------------------------------------------
     //Change log table:
     //Version       | Date          | Expert in charge      | Changes applied
     //----------------------------------------------------------------------------------------------------------
     //1.0.0         | 20.06.23      | HeitecAg                | First released Version
     //==========================================================================================================
   END_REGION BLOCK INFO HEADER


   REGION INIT

     #xlocalError := FALSE;
     #xSchrittketteTimeOut := FALSE;
     #fpCpuRestart(CLK := #iCpuRestart);

     //Sende Daten vom Bausteineingang einlesen
     #tempSendUserDaten[1] := #iUserDaten_iJaw1;
     #tempSendUserDaten[2] := #iUserDaten_iJaw2;
     #tempSendUserDaten[3] := #iUserDaten_iJaw3;
     #tempSendUserDaten[4] := #iUserDaten_iJaw4;
     #tempSendUserDaten[5] := #iUserDaten_iJaw5;
     #tempSendUserDaten[6] := #iUserDaten_iJaw6;
     #tempSendUserDaten[7] := #iUserDaten_iJaw7;
     #tempSendUserDaten[8] := #iUserDaten_iJaw8;

     //Flanke CPU Hochlauf
     IF #fpCpuRestart.Q
       OR #xlocalInit THEN
       #txFPCpuHochlauf := True;
       #xlocalInit := FALSE;
     ELSE
       #txFPCpuHochlauf := False;
     END_IF;



     //Überbrückung Hochlaufzeit Profinet
     #tonPNHochlaufzeit(IN := TRUE,
                        PT := #iTime_PnIoRyd);

     IF #txFPCpuHochlauf THEN

       #xlocalIoLinkRdy :=
       #xlocalIoLinkBusy :=
       #xlocalIoLinkError :=
       #xlocalFreeIsduCmdFertig :=
       #xlocalFreeIsduCmdDataBereit := FALSE;

       #iRetValLog2Geo := LOG2GEO(LADDR := #iLADDR_TigoMaster, GEOADDR := #tempHwInfoTigoMaster2Th);


       IF #iRetValLog2Geo = 0 THEN
         FOR #tdiI := 1 TO #MAX_HW_SLOTS DO

           #iRetValGeoLog[#tdiI] := GEO_LOG(MASTER := UINT_TO_INT(#tempHwInfoTigoMaster2Th.IOSYSTEM),
                                            STATION := UINT_TO_INT(#tempHwInfoTigoMaster2Th.STATION),
                                            SLOT := #SLOT_IDX_MAIN_MODUL_2TH,
                                            SUBSLOT := DINT_TO_INT(#tdiI),
                                            LADDR => #tempHwAny);

           IF (#iRetValGeoLog[#tdiI] = #KEIN_FEHLER)
             AND (#tempHwAny <> #DEF_HW_ANY) THEN
             #hwAnySubSlotsTigoMaster2Th[#tdiI] := #tempHwAny;
           ELSE
             #hwAnySubSlotsTigoMaster2Th[#tdiI] := #DEF_HW_ANY;
           END_IF;

         END_FOR;
       END_IF;

       #strIJawType[1] := #LEER_STRING;

       FOR #tdiI := 1 TO USINT_TO_DINT(#MAX_ANZAHL_IJAWS) DO
         #strIJawType[#tdiI] := #LEER_STRING;
         ;
       END_FOR;

     END_IF;

     #tempIJawAktiv[1] := #iIJawAktiv_iJaw1;
     #tempIJawAktiv[2] := #iIJawAktiv_iJaw2;
     #tempIJawAktiv[3] := #iIJawAktiv_iJaw3;
     #tempIJawAktiv[4] := #iIJawAktiv_iJaw4;
     #tempIJawAktiv[5] := #iIJawAktiv_iJaw5;
     #tempIJawAktiv[6] := #iIJawAktiv_iJaw6;
     #tempIJawAktiv[7] := #iIJawAktiv_iJaw7;
     #tempIJawAktiv[8] := #iIJawAktiv_iJaw8;

     REGION CHECK iJAW vorhanden

       #xMin1iJawVorh := FALSE;
       FOR #tdiI := 1 TO USINT_TO_DINT(#MAX_ANZAHL_IJAWS) DO

         IF #tempIJawAktiv[#tdiI]
           AND (#hwAnySubSlotsTigoMaster2Th[#tdiI] <> 0) THEN
           #arrIJawVorhandenAktiv[#tdiI] := TRUE;
           //Mindestens 1 iJaw vorhanden
           #xMin1iJawVorh := TRUE;
         ELSE
           #arrIJawVorhandenAktiv[#tdiI] := FALSE;
         END_IF;

       END_FOR;
     END_REGION CHECK iJAW vorhanden    

   END_REGION INIT

   REGION Profinet Slave aktivieren / deaktivieren
     //Reset bei Hochlauf
     IF #txFPCpuHochlauf THEN
       #strcDeaktAkt.ReqAkt := 0;
       #strcDeaktAkt.ReqDeak := 0;
       #strcDeaktAkt.IstAkt := 0;
       #strcDeaktAkt.IstDeak := 0;
       #strcDeaktAkt.ModNr := 0;
     END_IF;

     //Request PN Slave aktivieren
     IF #tonPNHochlaufzeit.Q AND #iPN_Act AND #xMin1iJawVorh AND NOT #txFPCpuHochlauf AND NOT #strcDeaktAkt.IstAkt THEN
       #strcDeaktAkt.ModNr := 1;
       #strcDeaktAkt.ReqAkt := TRUE;


     END_IF;

     //Request PN Slave deaktivieren
     IF #tonPNHochlaufzeit.Q AND (NOT #iPN_Act OR NOT #xMin1iJawVorh) AND NOT #txFPCpuHochlauf AND NOT #strcDeaktAkt.IstDeak THEN
       #strcDeaktAkt.ModNr := 2;
       #strcDeaktAkt.ReqDeak := TRUE;
       FOR #tdiI := 1 TO USINT_TO_DINT(#MAX_ANZAHL_IJAWS) DO
         #strIJawType[#tdiI] := #LEER_STRING;
         ;
       END_FOR;
     END_IF;

     #fpPnIOAktiv(CLK := #strcDeaktAkt.IstAkt);
     #fpPnIOInAktiv(CLK := #strcDeaktAkt.IstDeak);


     //Teilnehmer aktivieren / deaktivieren
     #strcDeaktAkt.Ret_Val := D_ACT_DP(REQ := #strcDeaktAkt.ReqAkt OR #strcDeaktAkt.ReqDeak, MODE := #strcDeaktAkt.ModNr, LADDR := #iLADDR_TigoMaster, BUSY => #strcDeaktAkt.busy);
     IF (#strcDeaktAkt.Ret_Val = 16#8090)
       OR (#strcDeaktAkt.Ret_Val = 16#8093)
       OR (#strcDeaktAkt.Ret_Val = 16#80a0)
       OR (#strcDeaktAkt.Ret_Val = 16#80a3)
       OR (#strcDeaktAkt.Ret_Val = 16#80a4)
       OR (#strcDeaktAkt.Ret_Val = 16#80c3)
     THEN
       #xlocalError := TRUE;
     END_IF;
     //Zustand Aktiviert / deaktiviert speichern
     //Trigger generieren
     IF #strcDeaktAkt.Ret_Val = 0 AND #strcDeaktAkt.ModNr <> 0 AND NOT #strcDeaktAkt.ChangeRequest_old THEN
       #strcDeaktAkt.FP_Changerequest := True;
     ELSE
       #strcDeaktAkt.FP_Changerequest := false;
     END_IF;
     #strcDeaktAkt.ChangeRequest_old := #strcDeaktAkt.Ret_Val = 0 AND #strcDeaktAkt.ModNr <> 0;

     //Status speicher
     //Slave ist aktiviert
     IF #strcDeaktAkt.FP_Changerequest AND #strcDeaktAkt.ModNr = 1 THEN
       #strcDeaktAkt.ReqAkt := 0;
       #strcDeaktAkt.ReqDeak := 0;
       #strcDeaktAkt.IstAkt := 1;
       #strcDeaktAkt.IstDeak := 0;
       #strcDeaktAkt.ModNr := 0;
       //Slave ist deaktiviert
     ELSIF #strcDeaktAkt.FP_Changerequest AND #strcDeaktAkt.ModNr = 2 THEN
       #strcDeaktAkt.ReqAkt := 0;
       #strcDeaktAkt.ReqDeak := 0;
       #strcDeaktAkt.IstAkt := 0;
       #strcDeaktAkt.IstDeak := 1;
       #strcDeaktAkt.ModNr := 0;
     END_IF;
   END_REGION

   REGION Daten Empfangen
     //Recive Data from iJaws 1..Anzahl iJaws
     //
     IF #xMin1iJawVorh AND #strcDeaktAkt.IstAkt THEN
       FOR #tdiI := 1 TO USINT_TO_DINT(#MAX_ANZAHL_IJAWS) DO

         IF (NOT #arrIJawVorhandenAktiv[#tdiI]) THEN
           CONTINUE;
         END_IF;

         //Empfangsbereich ablöschen
         FOR #tdiO := 1 TO #LAENGE_RCV_DATEN DO
           #tempRcvRohDaten[#tdiO] := 0;
         END_FOR;

         //Daten abholen wenn iJaw N vorhanden
         #iRetRcvData := DPRD_DAT(LADDR := #hwAnySubSlotsTigoMaster2Th[#tdiI + #HW_IDX_IO_LINK_MASTER], RECORD => #tempRcvRohDaten);
         IF #iRetRcvData <> 0 THEN
           #xlocalError := TRUE;
         END_IF;

         //Empfangene Daten aufbereiten
         #tempPosSer := 0;
         #iRetSer := Deserialize(SRC_ARRAY := #tempRcvRohDaten, DEST_VARIABLE => #tempRcvEinzelDaten, POS := #tempPosSer);
         IF #iRetSer <> 0 THEN
           #xlocalError := TRUE;
         END_IF;

         #tempRcvUserdaten[#tdiI].Gauge1 := WORD_TO_UINT(#tempRcvEinzelDaten.Gauge1);
         #tempRcvUserdaten[#tdiI].Gauge2 := WORD_TO_UINT(#tempRcvEinzelDaten.Gauge2);
         #tempRcvUserdaten[#tdiI].Battery := BYTE_TO_USINT(#tempRcvEinzelDaten.Battery);
         #tempRcvUserdaten[#tdiI].Temperature := BYTE_TO_SINT(#tempRcvEinzelDaten.Temperature);
         #tempRcvUserdaten[#tdiI].GyroXaxis := BYTE_TO_SINT(#tempRcvEinzelDaten.GyroXaxis);
         #tempRcvUserdaten[#tdiI].GyroYaxis := BYTE_TO_SINT(#tempRcvEinzelDaten.GyroYaxis);
         #tempRcvUserdaten[#tdiI].GyroZaxis := BYTE_TO_SINT(#tempRcvEinzelDaten.GyroZaxis);
         #tempRcvUserdaten[#tdiI].Force1 := WORD_TO_UINT(#tempRcvEinzelDaten.Force1);
         #tempRcvUserdaten[#tdiI].Force2 := WORD_TO_UINT(#tempRcvEinzelDaten.Force2);
       END_FOR;

     END_IF;

     #tempRcvUserdaten[1].iJawType := #strIJawType[1];
     #tempRcvUserdaten[2].iJawType := #strIJawType[2];
     #tempRcvUserdaten[3].iJawType := #strIJawType[3];
     #tempRcvUserdaten[4].iJawType := #strIJawType[4];
     #tempRcvUserdaten[5].iJawType := #strIJawType[5];
     #tempRcvUserdaten[6].iJawType := #strIJawType[6];
     #tempRcvUserdaten[7].iJawType := #strIJawType[7];
     #tempRcvUserdaten[8].iJawType := #strIJawType[8];



     //Empfangene Daten auf Bausteinausgang schreiben
     #oUserDaten_iJaw1 := #tempRcvUserdaten[1];
     #oUserDaten_iJaw2 := #tempRcvUserdaten[2];
     #oUserDaten_iJaw3 := #tempRcvUserdaten[3];
     #oUserDaten_iJaw4 := #tempRcvUserdaten[4];
     #oUserDaten_iJaw5 := #tempRcvUserdaten[5];
     #oUserDaten_iJaw6 := #tempRcvUserdaten[6];
     #oUserDaten_iJaw7 := #tempRcvUserdaten[7];
     #oUserDaten_iJaw8 := #tempRcvUserdaten[8];
   END_REGION

   REGION RESET FIFO PUFFER
     #fpResetIoLink(CLK := #iResetIoLinkKom);

     IF #txFPCpuHochlauf
       OR #fpResetIoLink.Q
       OR #fpPnIOAktiv.Q
       OR #fpPnIOInAktiv.Q
     THEN
       FOR #tdiI := 1 TO USINT_TO_DINT(#MAX_FIFO_IDX) DO
         #fifoPuffer[#tdiI] := #tempResetFifo;
         #usiLetzterFiFoEintrag := 0;
         #diAkuelleSchrittnr := #SCHRITT_RESET;
       END_FOR;
     END_IF;
   END_REGION RESET FIFO PUFFER

   REGION FIFO PUFFER IO-LINK KOMMANDOS
     IF #xMin1iJawVorh AND #strcDeaktAkt.IstAkt THEN

       #fpTriggerFreeISDU(CLK := #iFreeIsduCmd.execute);


       FOR #tdiI := 1 TO USINT_TO_DINT(#MAX_ANZAHL_IJAWS) DO

         #fpTriggerTara[#tdiI](CLK := #tempSendUserDaten[#tdiI].RelCmdTara);
         #fpTriggerSySMode[#tdiI](CLK := #tempSendUserDaten[#tdiI].RelCmdSysMode);
         #fpTriggerReadType[#tdiI](CLK := #tempSendUserDaten[#tdiI].RelReadType);
         #fpTriggerIMA[#tdiI](CLK := #tempSendUserDaten[#tdiI].RelIMA);
         #fpTriggerForceThreshold[#tdiI](CLK := #tempSendUserDaten[#tdiI].RelForceTreshold);
         #fpTriggerNoiseLevel[#tdiI](CLK := #tempSendUserDaten[#tdiI].RelNoiseLevel);
         #fpTriggerStoreToFlash[#tdiI](CLK := #tempSendUserDaten[#tdiI].RelStoreToFlash);




         IF #fpTriggerTara[#tdiI].Q AND #arrIJawVorhandenAktiv[#tdiI] THEN

           #usiLetzterFiFoEintrag += 1;
           #fifoPuffer[#usiLetzterFiFoEintrag].cmd := #CMD_TARA;
           #fifoPuffer[#usiLetzterFiFoEintrag].isuCmdData.execute := TRUE;
           #fifoPuffer[#usiLetzterFiFoEintrag].isuCmdData.readWrite := #WRITE;
           #fifoPuffer[#usiLetzterFiFoEintrag].isuCmdData."port" := DINT_TO_INT(#tdiI);
           #fifoPuffer[#usiLetzterFiFoEintrag].isuCmdData.index := #IDX_CMD_TARA;
           #fifoPuffer[#usiLetzterFiFoEintrag].isuCmdData.subindex := #SUB_IDX_CMD_TARA;
           #fifoPuffer[#usiLetzterFiFoEintrag].isuCmdData.writeLen := 1;

         END_IF;

         IF #fpTriggerSySMode[#tdiI].Q AND #arrIJawVorhandenAktiv[#tdiI] THEN
           #usiLetzterFiFoEintrag += 1;
           #fifoPuffer[#usiLetzterFiFoEintrag].cmd := #CMD_CHANGE_SYSMODE;
           #fifoPuffer[#usiLetzterFiFoEintrag].isuCmdData.execute := TRUE;
           #fifoPuffer[#usiLetzterFiFoEintrag].isuCmdData.readWrite := #WRITE;
           #fifoPuffer[#usiLetzterFiFoEintrag].isuCmdData."port" := DINT_TO_INT(#tdiI);
           #fifoPuffer[#usiLetzterFiFoEintrag].isuCmdData.index := #IDX_CMD_SYSMODE;
           #fifoPuffer[#usiLetzterFiFoEintrag].isuCmdData.subindex := #SUB_IDX_CMD_SYSMODE;
           #fifoPuffer[#usiLetzterFiFoEintrag].isuCmdData.writeLen := 1;
         END_IF;

         IF #fpTriggerReadType[#tdiI].Q AND #arrIJawVorhandenAktiv[#tdiI] THEN
           #usiLetzterFiFoEintrag += 1;
           #fifoPuffer[#usiLetzterFiFoEintrag].cmd := #CMD_READ_TYPE;
           #fifoPuffer[#usiLetzterFiFoEintrag].isuCmdData.execute := TRUE;
           #fifoPuffer[#usiLetzterFiFoEintrag].isuCmdData.readWrite := #READ;
           #fifoPuffer[#usiLetzterFiFoEintrag].isuCmdData."port" := DINT_TO_INT(#tdiI);
           #fifoPuffer[#usiLetzterFiFoEintrag].isuCmdData.index := #IDX_CMD_READ_TYPE;
           #fifoPuffer[#usiLetzterFiFoEintrag].isuCmdData.subindex := #SUB_IDX_CMD_READ_TYPE;
           #fifoPuffer[#usiLetzterFiFoEintrag].isuCmdData.writeLen := 0;
         END_IF;

         IF #fpTriggerIMA[#tdiI].Q AND #arrIJawVorhandenAktiv[#tdiI] THEN
           #usiLetzterFiFoEintrag += 1;
           #fifoPuffer[#usiLetzterFiFoEintrag].cmd := #CMD_APPLICATION_IMA;
           #fifoPuffer[#usiLetzterFiFoEintrag].isuCmdData.execute := TRUE;
           #fifoPuffer[#usiLetzterFiFoEintrag].isuCmdData.readWrite := #WRITE;
           #fifoPuffer[#usiLetzterFiFoEintrag].isuCmdData."port" := DINT_TO_INT(#tdiI);
           #fifoPuffer[#usiLetzterFiFoEintrag].isuCmdData.index := #IDX_CMD_APPLICATION_IMA;
           #fifoPuffer[#usiLetzterFiFoEintrag].isuCmdData.subindex := #SUB_IDX_CMD_APPLICATION_IMA;
           #fifoPuffer[#usiLetzterFiFoEintrag].isuCmdData.writeLen := 1;
         END_IF;

         IF #fpTriggerForceThreshold[#tdiI].Q AND #arrIJawVorhandenAktiv[#tdiI] THEN
           #usiLetzterFiFoEintrag += 1;
           #fifoPuffer[#usiLetzterFiFoEintrag].cmd := #CMD_FORCE_TRESHOLD;
           #fifoPuffer[#usiLetzterFiFoEintrag].isuCmdData.execute := TRUE;
           #fifoPuffer[#usiLetzterFiFoEintrag].isuCmdData.readWrite := #WRITE;
           #fifoPuffer[#usiLetzterFiFoEintrag].isuCmdData."port" := DINT_TO_INT(#tdiI);
           #fifoPuffer[#usiLetzterFiFoEintrag].isuCmdData.index := #IDX_CMD_FORCE_THRESHOLD;
           #fifoPuffer[#usiLetzterFiFoEintrag].isuCmdData.subindex := #SUB_IDX_CMD_FORCE_TRESHOLD;
           #fifoPuffer[#usiLetzterFiFoEintrag].isuCmdData.writeLen := 4;
         END_IF;

         IF #fpTriggerNoiseLevel[#tdiI].Q AND #arrIJawVorhandenAktiv[#tdiI] THEN
           #usiLetzterFiFoEintrag += 1;
           #fifoPuffer[#usiLetzterFiFoEintrag].cmd := #CMD_NOISE_LEVEL;
           #fifoPuffer[#usiLetzterFiFoEintrag].isuCmdData.execute := TRUE;
           #fifoPuffer[#usiLetzterFiFoEintrag].isuCmdData.readWrite := #WRITE;
           #fifoPuffer[#usiLetzterFiFoEintrag].isuCmdData."port" := DINT_TO_INT(#tdiI);
           #fifoPuffer[#usiLetzterFiFoEintrag].isuCmdData.index := #IDX_CMD_NOISE_LEVEL;
           #fifoPuffer[#usiLetzterFiFoEintrag].isuCmdData.subindex := #SUB_IDX_CMD_NOISE_LEVEL;
           #fifoPuffer[#usiLetzterFiFoEintrag].isuCmdData.writeLen := 2;
         END_IF;

         IF #fpTriggerStoreToFlash[#tdiI].Q AND #arrIJawVorhandenAktiv[#tdiI] THEN
           #usiLetzterFiFoEintrag += 1;
           #fifoPuffer[#usiLetzterFiFoEintrag].cmd := #CMD_STORE_TO_FLASH;
           #fifoPuffer[#usiLetzterFiFoEintrag].isuCmdData.execute := TRUE;
           #fifoPuffer[#usiLetzterFiFoEintrag].isuCmdData.readWrite := #WRITE;
           #fifoPuffer[#usiLetzterFiFoEintrag].isuCmdData."port" := DINT_TO_INT(#tdiI);
           #fifoPuffer[#usiLetzterFiFoEintrag].isuCmdData.index := #IDX_CMD_STORE_TO_FLASH;
           #fifoPuffer[#usiLetzterFiFoEintrag].isuCmdData.subindex := #SUB_IDX_SCMD_TORE_TO_FLASH;
           #fifoPuffer[#usiLetzterFiFoEintrag].isuCmdData.writeLen := 1;
         END_IF;

         IF #fpTriggerFreeISDU.Q
           AND (#iFreeIsduCmd."port" <=#MAX_ANZAHL_IJAWS)
           AND (#iFreeIsduCmd."port" >= 1)THEN
           IF #arrIJawVorhandenAktiv[#iFreeIsduCmd."port"] THEN
             #usiLetzterFiFoEintrag += 1;
             #fifoPuffer[#usiLetzterFiFoEintrag].cmd := #CMD_FREE_ISDU;
             #fifoPuffer[#usiLetzterFiFoEintrag].isuCmdData.execute := TRUE;
             #fifoPuffer[#usiLetzterFiFoEintrag].isuCmdData.readWrite := #iFreeIsduCmd.readWrite;
             #fifoPuffer[#usiLetzterFiFoEintrag].isuCmdData."port" := #iFreeIsduCmd."port";
             #fifoPuffer[#usiLetzterFiFoEintrag].isuCmdData.index := #iFreeIsduCmd.index;
             #fifoPuffer[#usiLetzterFiFoEintrag].isuCmdData.subindex := #iFreeIsduCmd.subindex;
             #fifoPuffer[#usiLetzterFiFoEintrag].isuCmdData.writeLen := #iFreeIsduCmd.writeLen;

             #xlocalFreeIsduCmdFertig := FALSE;
             #xlocalFreeIsduCmdDataBereit := FALSE;
             #oFreeIsduRcvData := #tempInitRecord;
           END_IF;
         END_IF;

       END_FOR;
     END_IF;
   END_REGION FIFO PUFFER IO-LINK KOMMANDOS

   REGION Schrittkette Kommandos schreiben

     IF #xMin1iJawVorh AND #strcDeaktAkt.IstAkt THEN
       // Statement section REGION
       CASE #diAkuelleSchrittnr OF

         #SCHRITT_RESET:

           (*IO-Link Status setzten*)
           #xlocalIoLinkRdy := FALSE;
           #xlocalIoLinkBusy := FALSE;
           #xlocalIoLinkError := FALSE;

           IF (#hwAnySubSlotsTigoMaster2Th[#HW_IDX_IO_LINK_MASTER] <> #DEF_HW_ANY) THEN
             #tempSchrittNr := #SCHRITT_CHECK_RDY;
             #txAktNächstenSchritt := TRUE;
             #strcIoLinkSignale.in.execute := FALSE;
           END_IF;

         #SCHRITT_CHECK_RDY:

           (*IO-Link Status setzten*)
           #xlocalIoLinkRdy := FALSE;
           #xlocalIoLinkBusy := FALSE;
           #xlocalIoLinkError := FALSE;

           IF (#strcDeaktAkt.IstAkt AND NOT #strcDeaktAkt.IstDeak)
             AND (NOT #strcIoLinkSignale.out.error)
             AND (#strcIoLinkSignale.out.status = 16#7000)
           THEN
             #tempSchrittNr := #SCHRITT_HOME;
             #txAktNächstenSchritt := TRUE;
           ELSIF (#strcIoLinkSignale.out.status = 16#8000)
             OR #strcIoLinkSignale.out.error
             AND (NOT #xSchrittErsterZyklus) THEN
             #tempSchrittNr := #SCHRITT_FEHLER;
             #txAktNächstenSchritt := TRUE;
           END_IF;

         #SCHRITT_HOME:

           (*IO-Link Status setzten*)
           #xlocalIoLinkRdy := TRUE;
           #xlocalIoLinkBusy := FALSE;
           #xlocalIoLinkError := FALSE;

           IF (#fifoPuffer[#IDX_FIFO_LESE_INDEX].cmd = #CMD_IDLE) THEN
             ;
           ELSIF (#fifoPuffer[#IDX_FIFO_LESE_INDEX].cmd = #CMD_TARA) THEN
             #tempSchrittNr := #SCHRITT_SEND_CMD;
             #txAktNächstenSchritt := TRUE;
           ELSIF (#fifoPuffer[#IDX_FIFO_LESE_INDEX].cmd = #CMD_CHANGE_SYSMODE) THEN
             #tempSchrittNr := #SCHRITT_SEND_CMD;
             #txAktNächstenSchritt := TRUE;
           ELSIF (#fifoPuffer[#IDX_FIFO_LESE_INDEX].cmd = #CMD_READ_TYPE) THEN
             #tempSchrittNr := #SCHRITT_SEND_CMD;
             #txAktNächstenSchritt := TRUE;
           ELSIF (#fifoPuffer[#IDX_FIFO_LESE_INDEX].cmd = #CMD_APPLICATION_IMA) THEN
             #tempSchrittNr := #SCHRITT_SEND_CMD;
             #txAktNächstenSchritt := TRUE;
           ELSIF (#fifoPuffer[#IDX_FIFO_LESE_INDEX].cmd = #"CMD_FORCE_TRESHOLD") THEN
             #tempSchrittNr := #SCHRITT_SEND_CMD;
             #txAktNächstenSchritt := TRUE;
           ELSIF (#fifoPuffer[#IDX_FIFO_LESE_INDEX].cmd = #CMD_NOISE_LEVEL) THEN
             #tempSchrittNr := #SCHRITT_SEND_CMD;
             #txAktNächstenSchritt := TRUE;
           ELSIF (#fifoPuffer[#IDX_FIFO_LESE_INDEX].cmd = #CMD_STORE_TO_FLASH) THEN
             #tempSchrittNr := #SCHRITT_SEND_CMD;
           ELSIF (#fifoPuffer[#IDX_FIFO_LESE_INDEX].cmd = #CMD_FREE_ISDU) THEN
             #tempSchrittNr := #SCHRITT_SEND_CMD;
             #txAktNächstenSchritt := TRUE;
           END_IF;

         #SCHRITT_SEND_CMD:

           (*IO-Link Status setzten*)
           #xlocalIoLinkRdy := FALSE;
           #xlocalIoLinkBusy := TRUE;
           #xlocalIoLinkError := FALSE;

           // Reset Record daten
           #strcIoLinkSignale.record := #tempInitRecord;

           #strcIoLinkSignale.in.execute := #fifoPuffer[#IDX_FIFO_LESE_INDEX].isuCmdData.execute;
           #strcIoLinkSignale.in."port" := #fifoPuffer[#IDX_FIFO_LESE_INDEX].isuCmdData."port";
           #strcIoLinkSignale.in.index := #fifoPuffer[#IDX_FIFO_LESE_INDEX].isuCmdData.index;
           #strcIoLinkSignale.in.subindex := #fifoPuffer[#IDX_FIFO_LESE_INDEX].isuCmdData.subindex;
           #strcIoLinkSignale.in.writeLen := #fifoPuffer[#IDX_FIFO_LESE_INDEX].isuCmdData.writeLen;
           #strcIoLinkSignale.in.readWrite := #fifoPuffer[#IDX_FIFO_LESE_INDEX].isuCmdData.readWrite;

           IF (#fifoPuffer[#IDX_FIFO_LESE_INDEX].cmd = #CMD_TARA) THEN
             #strcIoLinkSignale.record[0] := #RECORD_DATA_TARA;

           ELSIF (#fifoPuffer[#IDX_FIFO_LESE_INDEX].cmd = #CMD_CHANGE_SYSMODE) THEN
             #strcIoLinkSignale.record[0] := #tempSendUserDaten[#fifoPuffer[#IDX_FIFO_LESE_INDEX].isuCmdData."port"].Mode;

           ELSIF (#fifoPuffer[#IDX_FIFO_LESE_INDEX].cmd = #CMD_APPLICATION_IMA) THEN
             #strcIoLinkSignale.record[0] := USINT_TO_BYTE(#tempSendUserDaten[#fifoPuffer[#IDX_FIFO_LESE_INDEX].isuCmdData."port"].IMA);

           ELSIF (#fifoPuffer[#IDX_FIFO_LESE_INDEX].cmd = #CMD_FORCE_TRESHOLD) THEN
             #tempPosSer := 0;
             #iRetValWriteBig := WRITE_BIG(src_variable := #tempSendUserDaten[#fifoPuffer[#IDX_FIFO_LESE_INDEX].isuCmdData."port"].ForceTreshold,
                                           dest_array := #strcIoLinkSignale.record,
                                           pos := #tempPosSer);


           ELSIF (#fifoPuffer[#IDX_FIFO_LESE_INDEX].cmd = #CMD_NOISE_LEVEL) THEN
             #tempPosSer := 0;
             #iRetValWriteBig := WRITE_BIG(src_variable := #tempSendUserDaten[#fifoPuffer[#IDX_FIFO_LESE_INDEX].isuCmdData."port"].NoiseLevel,
                                           dest_array := #strcIoLinkSignale.record,
                                           pos := #tempPosSer);

           ELSIF (#fifoPuffer[#IDX_FIFO_LESE_INDEX].cmd = #CMD_STORE_TO_FLASH) THEN
             #strcIoLinkSignale.record[0] := #RECORD_STORE_TO_FLASH;

           ELSIF (#fifoPuffer[#IDX_FIFO_LESE_INDEX].cmd = #CMD_READ_TYPE) THEN
             ;

           ELSIF (#fifoPuffer[#IDX_FIFO_LESE_INDEX].cmd = #CMD_FREE_ISDU) THEN
             #strcIoLinkSignale.record := #iFreeIsduSendData;
           END_IF;

           IF #strcIoLinkSignale.out.error
             OR (#iRetValWriteBig <> 0) THEN
             #tempSchrittNr := #SCHRITT_FEHLER;
             #txAktNächstenSchritt := TRUE;
           ELSIF #strcIoLinkSignale.out.busy
             AND (NOT #strcIoLinkSignale.out.done) THEN
             #tempSchrittNr := #SCHRITT_WARTE_AUF_DONE;
             #txAktNächstenSchritt := TRUE;
           END_IF;

         #SCHRITT_WARTE_AUF_DONE:

           (*IO-Link Status setzten*)
           #xlocalIoLinkRdy := FALSE;
           #xlocalIoLinkBusy := TRUE;
           #xlocalIoLinkError := FALSE;

           IF #strcIoLinkSignale.out.done THEN

             IF (#fifoPuffer[#IDX_FIFO_LESE_INDEX].cmd = #CMD_READ_TYPE) THEN
               Chars_TO_Strg(Chars  := #strcIoLinkSignale.record,
                             pChars := #P_CHAR_CONV_STRING,
                             Cnt    := #CNT_CONV_STRING,
                             Strg   => #strIJawType[#fifoPuffer[#IDX_FIFO_LESE_INDEX].isuCmdData."port"]);

             ELSIF (#fifoPuffer[#IDX_FIFO_LESE_INDEX].cmd = #CMD_FREE_ISDU) THEN

               #xlocalFreeIsduCmdFertig := TRUE;
               #oFreeIsduRcvData := #tempInitRecord;

               IF (#fifoPuffer[#IDX_FIFO_LESE_INDEX].isuCmdData.readWrite = #READ) THEN
                 #xlocalFreeIsduCmdDataBereit := TRUE;
                 #recordDataFreeISDU := #strcIoLinkSignale.record;
               ELSE
                 #xlocalFreeIsduCmdDataBereit := FALSE;
               END_IF;

             END_IF;

             #strcIoLinkSignale.in.execute := FALSE;
             #tempSchrittNr := #SCHRITT_BEARBEITE_FIFO;
             #txAktNächstenSchritt := TRUE;
           ELSIF #strcIoLinkSignale.out.error THEN
             #tempSchrittNr := #SCHRITT_FEHLER;
             #txAktNächstenSchritt := TRUE;
           END_IF;


         #SCHRITT_BEARBEITE_FIFO:

           (*IO-Link Status setzten*)
           #xlocalIoLinkRdy := FALSE;
           #xlocalIoLinkBusy := TRUE;
           #xlocalIoLinkError := FALSE;

           FOR #tdiO := USINT_TO_DINT(#usiLetzterFiFoEintrag) TO 1 BY -1 DO
             IF (#tdiO = 1) THEN
               #fifoPuffer[#tdiO] := #tempResetFifo;
               #usiLetzterFiFoEintrag += -1;
             ELSIF
               (#tdiO <= USINT_TO_DINT(#MAX_FIFO_IDX))
               AND (#tdiO > 1) THEN
               #fifoPuffer[#tdiO - 1] := #fifoPuffer[#tdiO];
               #fifoPuffer[#tdiO] := #tempResetFifo;
               #usiLetzterFiFoEintrag += -1;
             ELSE
               EXIT;
             END_IF;
           END_FOR;

           #tempSchrittNr := #SCHRITT_CHECK_RDY;
           #txAktNächstenSchritt := TRUE;

         #SCHRITT_FEHLER:

           (*IO-Link Status setzten*)
           #xlocalIoLinkRdy := FALSE;
           #xlocalIoLinkBusy := FALSE;
           #xlocalIoLinkError := TRUE;

           #xSchrittketteTimeOut := TRUE;
           #xlocalError := TRUE;

           IF #iAck_Fehler_IoLinkKom THEN

             #strcIoLinkSignale.in.execute := FALSE;

             #tempSchrittNr := #SCHRITT_CHECK_RDY;
             #txAktNächstenSchritt := TRUE;
           END_IF;

         ELSE  // Statement section ELSE
           ;
       END_CASE;

       REGION SCHRITT UMSCHALTUNG
         #xSchrittErsterZyklus := FALSE;

         IF #txAktNächstenSchritt
           AND (#tempSchrittNr >= #SCHRITT_CHECK_RDY)
           AND (#tempSchrittNr <= #SCHRITT_FEHLER) THEN
           #diUrAlteSchrittnr := #diAlteSchrittnr;
           #diAlteSchrittnr := #diAkuelleSchrittnr;
           #diAkuelleSchrittnr := #tempSchrittNr;
           #xSchrittErsterZyklus := TRUE;
         END_IF;

         REGION SCHRITTZEIT
           #iRetValCpuZeitLesen := RD_SYS_T(#dtCpuSystemDatumZeit);
           #todCpuSystemZeit := DT_TO_TOD(#dtCpuSystemDatumZeit);
           #tCpuSystemZeit := TOD_TO_TIME(#todCpuSystemZeit);

           IF #xSchrittErsterZyklus
             OR (#tAktuelleSchrittzeit >= #MAX_TIME) THEN
             #tStartZeitSchritt := #tCpuSystemZeit;
             #tSchrittZeitVortag := #DEAK_SCHRITT_ZEIT_UEBERW;
           ELSIF (#todCpuSystemZeit = #DEF_TIME_OF_DAY) THEN
             #tSchrittZeitVortag := #tAktuelleSchrittzeit;
             #tStartZeitSchritt := #tCpuSystemZeit;
           END_IF;

           #tAktuelleSchrittzeit := (#tCpuSystemZeit - #tStartZeitSchritt) + #tSchrittZeitVortag;

           IF (#tMaxSchrittZeit > #DEAK_SCHRITT_ZEIT_UEBERW)
             AND (#tMaxSchrittZeit > #tAktuelleSchrittzeit)
           THEN
             #xFehlerSchrittZeitUeberwachung := TRUE;
           ELSE
             #xFehlerSchrittZeitUeberwachung := FALSE;
           END_IF;

         END_REGION SCHRITTZEIT


       END_REGION SCHRITT UMSCHALTUNG
     ELSE
       #xlocalIoLinkRdy := FALSE;
       #xlocalIoLinkBusy := FALSE;
       #xlocalIoLinkError := FALSE;

     END_IF;

   END_REGION

   REGION BEREITSTELLUNG RCV DATEN FREE ISDU-AUFTRAG
     IF #iFreeIsduCmd.execute
       AND (#strcDeaktAkt.IstAkt AND NOT #strcDeaktAkt.IstDeak)
     THEN
       IF #xlocalFreeIsduCmdFertig
         AND #xlocalFreeIsduCmdDataBereit
       THEN
         #oFreeIsduRcvData := #recordDataFreeISDU;
       END_IF;
     ELSE
       #xlocalFreeIsduCmdFertig := FALSE;
       #xlocalFreeIsduCmdDataBereit := FALSE;
       #oFreeIsduRcvData := #recordDataFreeISDU := #tempInitRecord;
     END_IF;
   END_REGION BEREITSTELLUNG RCV DATEN FREE ISDU-AUFTRAG


   REGION AUFRUF IO_LINK DEVICE

     REGION INIT IO-Link
       #strcIoLinkSignale.in.hwID := #hwAnySubSlotsTigoMaster2Th[#HW_IDX_IO_LINK_MASTER];
       #strcIoLinkSignale.in.cap := #CAP_IOLINK;
     END_REGION INIT IO-Link 

     #instLIOLinkDev(execute       := #strcIoLinkSignale.in.execute,
                     hwID          := #strcIoLinkSignale.in.hwID,
                     cap           := #strcIoLinkSignale.in.cap,
                     readWrite     := #strcIoLinkSignale.in.readWrite,
                     "port"        := #strcIoLinkSignale.in."port",
                     index         := #strcIoLinkSignale.in.index,
                     subindex      := #strcIoLinkSignale.in.subindex,
                     writeLen      := #strcIoLinkSignale.in.writeLen,
                     timeout       := #strcIoLinkSignale.in.timeout,
                     pollingPeriod := #strcIoLinkSignale.in.pollingPeriod,
                     done          => #strcIoLinkSignale.out.done,
                     busy          => #strcIoLinkSignale.out.busy,
                     error         => #strcIoLinkSignale.out.error,
                     status        => #strcIoLinkSignale.out.status,
                     diagnostics   => #strcIoLinkSignale.out.diagnostics,
                     readLen       => #strcIoLinkSignale.out.readLen,
                     record        := #strcIoLinkSignale.record);

     #wErrorW0 := #strcIoLinkSignale.out.diagnostics.subfunctionStatus.%W0;
     #wErrorW1 := #strcIoLinkSignale.out.diagnostics.subfunctionStatus.%W1;


   END_REGION AUFRUF IO_LINK DEVICE

   REGION Daten senden
     //Daten senden an iJaw 1..Anzahl iJaws

     IF #xMin1iJawVorh AND #strcDeaktAkt.IstAkt THEN

       //Daten aufbereiten
       FOR #tdiI := 1 TO USINT_TO_DINT(#MAX_ANZAHL_IJAWS) DO
         IF (NOT #arrIJawVorhandenAktiv[#tdiI]) THEN
           CONTINUE;
         END_IF;

         //wenn iJaw vorhanden
         #tempSendDaten.nRotSpeedSpindleAct := #tempSendUserDaten[#tdiI].nRotSpeedSpindleAct;
         #tempSendDaten.pHydCylChamber1Act := #tempSendUserDaten[#tdiI].pHydCylChamber1Act;
         #tempSendDaten.pHydCylChamber2Act := #tempSendUserDaten[#tdiI].pHydCylChamber2Act;
         #tempSendDaten.AHydCylChamber1Act := #tempSendUserDaten[#tdiI].AHydCylChamber1Act;
         #tempSendDaten.AHydCylChamber2Act := #tempSendUserDaten[#tdiI].AHydCylChamber2Act;

         //Daten senden
         IF #strcDeaktAkt.IstAkt THEN
           #iRetSendData := DPWR_DAT(LADDR := #hwAnySubSlotsTigoMaster2Th[#tdiI + #HW_IDX_IO_LINK_MASTER], RECORD := #tempSendDaten);
           IF #iRetSendData <> 0 THEN
             #xlocalError := TRUE;
           END_IF;
         END_IF;
       END_FOR;
     END_IF;
   END_REGION

   REGION BAUSTEIN ENDE
     #oIoLinkRdy := #xlocalIoLinkRdy;
     #oIoLinkBusy := #xlocalIoLinkBusy;
     #oIoLinkError := #xlocalIoLinkError;

     #oFreeIsduCmdFertig := #xlocalFreeIsduCmdFertig;
     #oFreeIsduCmdDataBereit := #xlocalFreeIsduCmdDataBereit;

     // Setze Bausteinausgang Teilnehmer aktiv
     #oPnTeilAkt := #strcDeaktAkt.IstAkt AND NOT #strcDeaktAkt.IstDeak;

     #oError := #xlocalError;
     ENO := (NOT #xlocalError);
     RETURN;
   END_REGION BAUSTEIN ENDE
END_FUNCTION_BLOCK

